(* Logix 5000 project; controller ODSI_Testing vendor 1 type 14 code 151 rev 20.19; software revision 20.05 *)

TASK MainTask (continuous, watchdog 500 ms) : MainProgram

MODULES
   Local : vendor 1 type 14 code 151 (Compact 0, rev 20.19)
      Counters : Embedded (Compact 3, rev 1.1, Output RPI 20 ms)
      Discrete_IO : Embedded (Compact 1, rev 3.1, Output RPI 20 ms)
      ASCII_1 : vendor 1 type 109 code 66 (Compact 5, rev 2.1, Output RPI 2 ms)
      Analog_IO : Embedded (Compact 2, rev 1.1, Output RPI 80 ms)
      OW16_1 : 1769-OW16 (Compact 4, rev 1.1, Output RPI 20 ms)
END_MODULES

VAR_GLOBAL   (* controller tags *)
   HMI_Stop : BOOL;
   ODSI_Valve1 : ALIAS FOR Local:1:I.Data.0;
   ODSI_Valve2 : ALIAS FOR Local:1:I.Data.1;
   ODSI_Valve3 : ALIAS FOR Local:1:I.Data.2;
   OSDI_Fail_Sample1 : ALIAS FOR Local:1:I.Data.4;
   OSDI_Fail_Sample2 : ALIAS FOR Local:1:I.Data.6;
   OSDI_Fail_Sample3 : ALIAS FOR Local:1:I.Data.8;
   OSDI_Pass_Sample1 : ALIAS FOR Local:1:I.Data.3;
   OSDI_Pass_Sample2 : ALIAS FOR Local:1:I.Data.5;
   OSDI_Pass_Sample3 : ALIAS FOR Local:1:I.Data.7;
   Request_Delay : DINT := 10;
   S1_PB_Input : BOOL;
   S1_Request : ALIAS FOR Local:1:O.Data.0;
   S1_Request_Delay : TIMER := (PRE := 10000);
   S2_PB_Input : BOOL;
   S2_Request : ALIAS FOR Local:1:O.Data.1;
   S2_Request_Delay : TIMER := (PRE := 10000);
   S3_PB_Input : BOOL;
   S3_Request : ALIAS FOR Local:1:O.Data.2;
   S3_Request_Delay : TIMER := (PRE := 10000);
   Valve1_Open : ALIAS FOR Local:1:O.Data.3;
   Valve1_Open_Delay : TIMER := (PRE := 10000);
   Valve2_Open : ALIAS FOR Local:1:O.Data.4;
   Valve2_Open_Delay : TIMER := (PRE := 10000);
   Valve3_Open : ALIAS FOR Local:1:O.Data.5;
   Valve3_Open_Delay : TIMER := (PRE := 10000);
   Valve_Block : BOOL := 1;
   Valve_Delay : DINT := 10;
END_VAR

PROGRAM MainProgram   (* main routine MainRoutine *)

ROUTINE MainRoutine   (* ladder *)
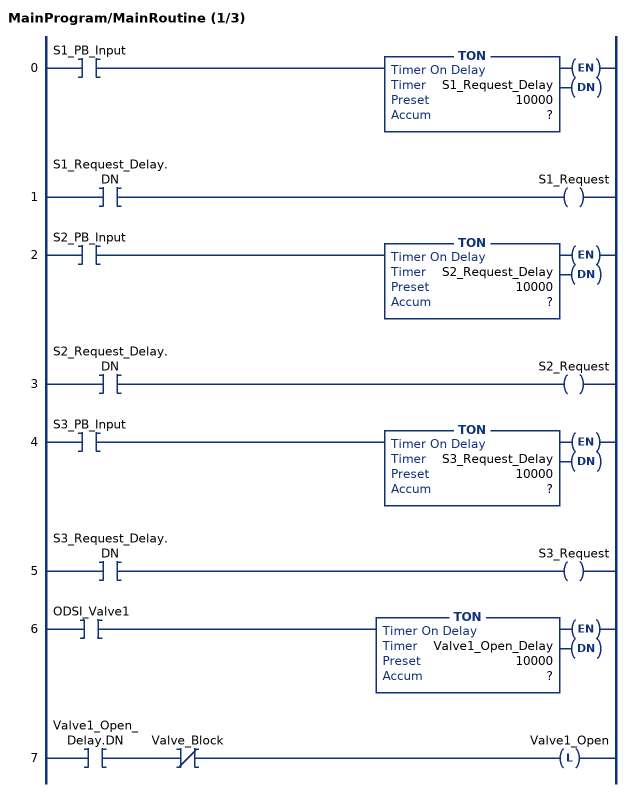
   0: XIC(S1_PB_Input)TON(S1_Request_Delay,?,?);
   1: XIC(S1_Request_Delay.DN)OTE(S1_Request);
   2: XIC(S2_PB_Input)TON(S2_Request_Delay,?,?);
   3: XIC(S2_Request_Delay.DN)OTE(S2_Request);
   4: XIC(S3_PB_Input)TON(S3_Request_Delay,?,?);
   5: XIC(S3_Request_Delay.DN)OTE(S3_Request);
   6: XIC(ODSI_Valve1)TON(Valve1_Open_Delay,?,?);
   7: XIC(Valve1_Open_Delay.DN)XIO(Valve_Block)OTL(Valve1_Open);
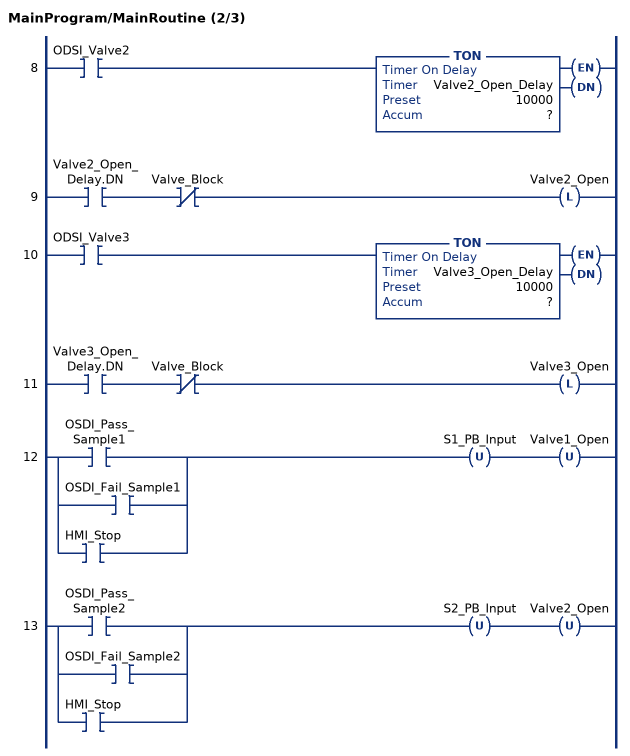
   8: XIC(ODSI_Valve2)TON(Valve2_Open_Delay,?,?);
   9: XIC(Valve2_Open_Delay.DN)XIO(Valve_Block)OTL(Valve2_Open);
   10: XIC(ODSI_Valve3)TON(Valve3_Open_Delay,?,?);
   11: XIC(Valve3_Open_Delay.DN)XIO(Valve_Block)OTL(Valve3_Open);
   12: [XIC(OSDI_Pass_Sample1) ,XIC(OSDI_Fail_Sample1) ,XIC(HMI_Stop) ]OTU(S1_PB_Input)OTU(Valve1_Open);
   13: [XIC(OSDI_Pass_Sample2) ,XIC(OSDI_Fail_Sample2) ,XIC(HMI_Stop) ]OTU(S2_PB_Input)OTU(Valve2_Open);
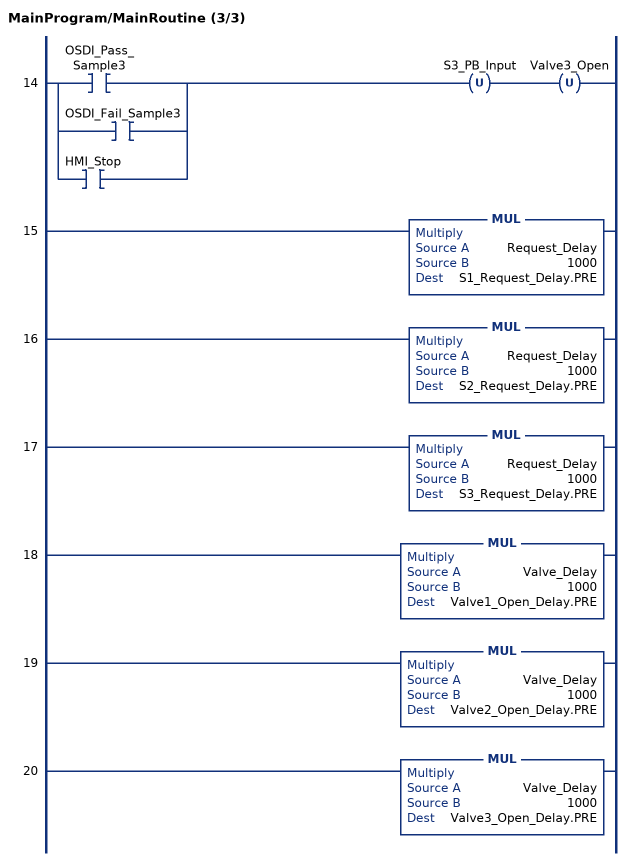
   14: [XIC(OSDI_Pass_Sample3) ,XIC(OSDI_Fail_Sample3) ,XIC(HMI_Stop) ]OTU(S3_PB_Input)OTU(Valve3_Open);
   15: MUL(Request_Delay,1000,S1_Request_Delay.PRE);
   16: MUL(Request_Delay,1000,S2_Request_Delay.PRE);
   17: MUL(Request_Delay,1000,S3_Request_Delay.PRE);
   18: MUL(Valve_Delay,1000,Valve1_Open_Delay.PRE);
   19: MUL(Valve_Delay,1000,Valve2_Open_Delay.PRE);
   20: MUL(Valve_Delay,1000,Valve3_Open_Delay.PRE);
END_ROUTINE
END_PROGRAM
